FUNCTION F_FormatString5 : T_MaxString
VAR_INPUT
	Format	: T_MaxString;
	arg1	: T_Arg;
	arg2	: T_Arg;
	arg3	: T_Arg;
	arg4	: T_Arg;
	arg5	: T_Arg;
END_VAR
VAR
    FB_FormatString1 : FB_FormatString;
END_VAR

FB_FormatString1(
	sFormat:= Format, 
	arg1:= arg1, 
	arg2:= arg2, 
	arg3:= arg3, 
	arg4:= arg4, 
	arg5:= arg5, 
	arg6:= , 
	arg7:= , 
	arg8:= , 
	arg9:= , 
	arg10:= , 
	bError=> , 
	nErrId=> , 
	sOut=> F_FormatString5);

END_FUNCTION

(* stored: Version 1.1.0.1, ProductVersion 3.1.4024.3
   POU F_FormatString5: Id {8194dfe8-2021-4048-a397-f5532b9c3378}, SpecialFunc None *)
